TYPE TupleStruct_1:
    STRUCT
        field1: TupleStruct;
        field2: LREAL;
    END_STRUCT
END_TYPE

(* stored: ProductVersion 3.1.0.18, Version 1.1.0.1 *)
